// TwinCAT 3 PLC project MainProgram
// ProgramVersion: 3.1.4023.0
// libraries:
//   Tc2_Standard, * (Beckhoff Automation GmbH)
//   Tc2_System, * (Beckhoff Automation GmbH)
//   Tc2_Utilities, * (Beckhoff Automation GmbH)
//   Tc3_Module, * (Beckhoff Automation GmbH)
// project tree:
//   / PlcTask.TcTTO
//   POUs/ MAIN.TcPOU
// real-time tasks:
//   TASK PlcTask: cycle T#10ms, priority 20, ADS port 350

CONFIGURATION MainProgram
    RESOURCE PLC ON TwinCAT3
        TASK PlcTask(INTERVAL := T#10ms, PRIORITY := 20);
        PROGRAM MAIN WITH PlcTask : MAIN;
    END_RESOURCE
END_CONFIGURATION

// ---- POUs/MAIN.TcPOU
PROGRAM MAIN
VAR
	trigger : BOOL := TRUE;
	createGuid : FB_CreateGuid;
	guid : GUID;
	guidAsString : STRING;
END_VAR

IF NOT createGuid.bBusy AND trigger THEN	
	
	trigger := FALSE;
	createGuid(bExecute := FALSE);	
	createGuid(
			bExecute := TRUE,
			pGuidBuffer := ADR(guid),
			nGuidBufferSize := SIZEOF(guid));
			
ELSIF createGuid.bBusy THEN
	
	createGuid();	
	
END_IF

// The code abover this point does not require any further libraries.  
// ------------------------------------------------------------------
// The code below requires Tc2_Utilites

guidAsString := GUID_TO_STRING(guid);

END_PROGRAM
